{attribute addProperty BoxType "EK1960-0000-0021"}
{attribute addProperty Id "FSOEAT %Q*FSOE_B358BD5C12015"}
{attribute addProperty CRC "3675236599"}
{attribute addProperty SizeInBites "120"}
{attribute addProperty SizeInBytes "15"}
TYPE FSoE_Outputs_DB0FA8F7 :
STRUCT
	{attribute addProperty Name "FSOE"}
	FSOE AT %Q* : FSOE_B358BD5C;
END_STRUCT
END_TYPE

(* stored: Version 1.2.0.0, ProductVersion 3.1.4024.9
   DUT FSoE_Outputs_DB0FA8F7: Id {20e69ccf-8c2e-4d67-9134-abde8892d011} *)
